// TIA Portal V20 export
FUNCTION "StepToString" : String   // FC33, SCL
// stored: Namespace Unit1.Em2, SetENOAutomatically false
   VAR_INPUT
      StepDINT : DInt;   // DINT value of the step
   END_VAR
BEGIN
   // Translates the sequence step number to the step name
   // Adjusted for Sequence_1_SemiAutoSplice real use case

   CASE #StepDINT OF
       1:
           #StepToString := 'Idle';

       101:
           #StepToString := 'Tape Attach Unit HomePos Check';
       111:
           #StepToString := 'Tape Loading Turn HomePos Check';

       201:
           #StepToString := 'UW Semi Splicer Vacuum ALL HomePos Check';
       211:
           #StepToString := 'Electrode Cutter HomePos Check';
       221:
           #StepToString := 'Electrode Fix ALL HomePos Check';
       231:
           #StepToString := 'Electrode Fix Left Top Up & Left Bottom Down Check';
       241:
           #StepToString := 'Stopper HomePos Check';

       301:
           #StepToString := 'Splicing L/R Module Mover WorkPos Check';
       303:
           #StepToString := 'Electrode Holder Mover HomePos Check';
       311:
           #StepToString := 'Support Unit Shaft Pos Check';
       321:
           #StepToString := 'Frame Cover Pos Check';
       331:
           #StepToString := 'Support Unit Transfer HomePos Check';
       341:
           #StepToString := 'Support Unit Shaft WorkPos Check';
       351:
           #StepToString := 'Frame Cover WorkPos Check';

       401:
           #StepToString := 'Splicing L/R Module Mover HomePos Check';
       403:
           #StepToString := 'Electrode Holder Mover HomePos Check';
       411:
           #StepToString := 'Support Unit Shaft Pos Check';
       421:
           #StepToString := 'Frame Cover Pos Check';
       431:
           #StepToString := 'Support Unit Transfer WorkPos Check';
       441:
           #StepToString := 'Support Unit Shaft HomePos Check';
       451:
           #StepToString := 'Frame Cover WorkPos Check';

       501:
           #StepToString := 'Splicing Module Mover WorkPos Command';

       701:
           #StepToString := 'Stopper WorkPos Command';
       711:
           #StepToString := 'Electrode Fix Left Top Down & Bottom Up Command';
       721:
           #StepToString := 'Electrode Fix ALL WorkPos Command';
       731:
           #StepToString := 'UW Semi Splicer Vacuum All WorkPos Command';

       801:
           #StepToString := 'Electrode Cutter WorkPos Command';
       811:
           #StepToString := 'Electrode Cutter HomePos Command';

       901:
           #StepToString := 'Vacuum LB & RT HomePos Command';
       911:
           #StepToString := 'Unwinder Left Rewinding & Right Holder Home';
       921:
           #StepToString := 'Vacuum LT HomePos & RT WorkPos Command';

       1001:
           #StepToString := 'Vacuum LT & RB HomePos Command';
       1011:
           #StepToString := 'Unwinder Right Rewinding & Left Holder Home';
       1021:
           #StepToString := 'Vacuum LB HomePos & RB WorkPos Command';

       1101:
           #StepToString := 'Electrode Fix Left Top & Bottom HomePos';
       1111:
           #StepToString := 'Electrode Fix Left Top Up & Bottom HomePos';
       1121:
           #StepToString := 'Tape Loading Turn WorkPos Command';

       1201:
           #StepToString := 'Tape Attach Unit WorkPos Command';
       1211:
           #StepToString := 'UW Semi Splicer Tape Vacuum HomePos Command';
       1221:
           #StepToString := 'Tape Attach Unit HomePos Command';

       1301:
           #StepToString := 'Tape Loading Turn HomePos Command';
       1311:
           #StepToString := 'Vacuum Right Top & Bottom HomePos Command';
       1321:
           #StepToString := 'Electrode Fix Right Top & Bottom HomePos';
       1331:
           #StepToString := 'Stopper HomePos Command';
       1341:
           #StepToString := 'EM Link Change Check';
       1345:
           #StepToString := 'EM Link Change Left -> Right Command';
       1346:
           #StepToString := 'EM Link Change Right -> Left Command';
       1348:
           #StepToString := 'EM Link Change Complete';

       1401:
           #StepToString := 'Splicing Left Module Mover HomePos Command';
       1411:
           #StepToString := 'Support Unit Shaft HomePos Command';
       1413:
           #StepToString := 'Frame Cover HomePos Command';
       1421:
           #StepToString := 'Support Unit Transfer WorkPos Command LH->RH';
       1423:
           #StepToString := 'Frame Cover WorkPos Command';
       1431:
           #StepToString := 'Support Unit Shaft WorkPos Command';

       1501:
           #StepToString := 'Splicing Right Module Mover HomePos Command';
       1511:
           #StepToString := 'Support Unit Shaft HomePos Command';
       1513:
           #StepToString := 'Frame Cover HomePos Command';
       1521:
           #StepToString := 'Support Unit Transfer HomePos Command LH<-RH';
       1523:
           #StepToString := 'Frame Cover WorkPos Command';
       1531:
           #StepToString := 'Support Unit Shaft WorkPos Command';

       2001:
           #StepToString := 'Splicing Module Mover WorkPos Command';
       2004:
           #StepToString := 'Stopper WorkPos Command';
       2007:
           #StepToString := 'Electrode Fix Top Down & Bottom Up Command';
       2010:
           #StepToString := 'Electrode Fix ALL WorkPos Command';
       2013:
           #StepToString := 'UW Semi Splicer Vacuum All WorkPos Command';
       2016:
           #StepToString := 'Electrode Cutter WorkPos Command';
       2019:
           #StepToString := 'Electrode Cutter HomePos Command';
       2022:
           #StepToString := 'Vacuum Bottom & Top HomePos Command';
       2025:
           #StepToString := 'Unwinder Rewinding & Electrode Holder Home';
       2028:
           #StepToString := 'Vacuum Top HomePos & Top WorkPos Command';
       2031:
           #StepToString := 'Electrode Fix Top & Bottom HomePos Command';
       2034:
           #StepToString := 'Electrode Fix Top & Bottom HomePos Command';
       2037:
           #StepToString := 'Tape Loading Turn WorkPos Command';
       2040:
           #StepToString := 'Tape Attach Unit WorkPos Command';
       2043:
           #StepToString := 'UW Semi Splicer Tape Vacuum HomePos Command';
       2046:
           #StepToString := 'Tape Attach Unit HomePos Command';
       2049:
           #StepToString := 'Tape Loading Turn HomePos Command';
       2052:
           #StepToString := 'Vacuum Top & Bottom HomePos Command';
       2055:
           #StepToString := 'Electrode Fix Top & Bottom HomePos Command';
       2058:
           #StepToString := 'Stopper HomePos Command';
       2061:
           #StepToString := 'EM Link Change Check';
       2064:
           #StepToString := 'EM Link Change EM0 -> EM1 Command';
       2067:
           #StepToString := 'EM Link Change EM1 -> EM2 Command';
       2070:
           #StepToString := 'EM Link Change Complete';
       2073:
           #StepToString := 'Splicing Module Mover HomePos Command';
       2076:
           #StepToString := 'Support Unit Shaft HomePos Command';
       2079:
           #StepToString := 'Frame Cover HomePos Command';
       2082:
           #StepToString := 'Support Unit Transfer WorkPos Command LH<->RH';
       2085:
           #StepToString := 'Frame Cover WorkPos Command';
       2088:
           #StepToString := 'Support Unit Shaft WorkPos Command';

       9001:
           #StepToString := 'Immediate Stop';

       ELSE
           #StepToString := 'N/A';

   END_CASE;
END_FUNCTION
